PROGRAM MAIN
VAR
END_VAR

END_PROGRAM

(* stored: Version 1.1.0.1
   POU MAIN: Id {4ef65e4f-3fc3-4b8d-9082-32ff912527e7} *)
